TYPE TLoaderSynchro :
	(LS_TableLeftPart1 := 0,LS_TableLeftPart2,LS_TableRightPart1,LS_TableRightPart2,LS_END);
END_TYPE

(* stored: Version 1.1.0.1, ProductVersion 3.1.4022.12
   DUT TLoaderSynchro: Id {aac3e0bb-9f8f-45e8-955a-8a5c591f035e} *)
